Staubli VAL3: s2s7En.pjx

--- s2s7En.pjx ---
Parameters version=s7.9.1 stackSize=5000 millimeterUnit=true
Program file=connectTo.pgx
Program file=getBitAt.pgx
Program file=getByteAt.pgx
Program file=getDBsize.pgx
Program file=getdWordAt.pgx
Program file=getWordAt.pgx
Program file=init.pgx
Program file=ISOConnect.pgx
Program file=isoPDUsize.pgx
Program file=NegotPduLength.pgx
Program file=readArea.pgx
Program file=readDB.pgx
Program file=readme.pgx
Program file=recvISOpacket.pgx
Program file=recvPacket.pgx
Program file=sendPacket.pgx
Program file=setBitAt.pgx
Program file=setByteAt.pgx
Program file=setLastError.pgx
Program file=setWordAt.pgx
Program file=TCPConnect.pgx
Program file=writeArea.pgx
Data file=s2s7En.dtx
Library alias=bitOp path=./Binary7En/Binary7En.pjx
Type name=ISO_PDU_DATA_T path=./ISO_PDU_DATA_T/ISO_PDU_DATA_T.pjx

--- s2s7En.dtx ---
ISO_PDU_DATA_T PDU
  [0]
    num COPT[3]
    S7telegram_T S7telegram
      [0]
        num DATA[240]
        num H[18]
    num TPKT[4]
bool bConnected
public num nAreaCT = 28
public num nAreaDB = 132
public num nAreaMK = 131
public num nAreaPA = 130
public num nAreaPE = 129
public num nAreaTM = 29
num nCC = 208
num nConnType
num nDataBuffer[500]
num nDataSize
num nErrDataRead = 768
num nErrDataWrite = 1024
num nErrISOConnFail = 6
num nErrISOInvPDU = 8
num nErrISONegPDU = 7
num nErrS7Func = 1280
num nErrTCPConnRst = 2
num nErrTCPSend = 4
num nISOPort = 102
num nISO_CR[22]
  [0] = 3
  [3] = 22
  [4] = 17
  [5] = 224
  [9] = 1
  [11] = 192
  [12] = 1
  [13] = 10
  [14] = 193
  [15] = 2
  [16] = 1
  [18] = 194
  [19] = 2
  [20] = 1
  [21] = 2
num nISOheaderSize = 7
public num nLastError
num nLastPDUType
num nLocalTSAP_HI
num nLocalTSAP_LO
num nMaxPduSize = 247
num nMinPduSize = 16
public num nNoErrors
num nPDULength
num nRDsize = 31
num nRecvTimeout = 0.5
num nRemoteTSAP_HI
num nRemoteTSAP_LO
num nS7WLCounter = 28
num nS7WLTimer = 29
num nS7_BI[37]
  [0] = 3
  [3] = 37
  [4] = 2
  [5] = 240
  [6] = 128
  [7] = 50
  [8] = 7
  [11] = 5
  [14] = 8
  [16] = 12
  [18] = 1
  [19] = 18
  [20] = 4
  [21] = 17
  [22] = 67
  [23] = 3
  [25] = 255
  [26] = 9
  [28] = 8
  [29] = 48
  [30] = 65
  [31] = 48
  [32] = 48
  [33] = 48
  [34] = 48
  [35] = 48
  [36] = 65
num nS7_PN[25]
  [0] = 3
  [3] = 25
  [4] = 2
  [5] = 240
  [6] = 128
  [7] = 50
  [8] = 1
  [11] = 4
  [14] = 8
  [17] = 240
  [20] = 1
  [22] = 1
  [24] = 240
num nS7_R[31]
  [0] = 3
  [3] = 31
  [4] = 2
  [5] = 240
  [6] = 128
  [7] = 50
  [8] = 1
  [11] = 5
  [14] = 14
  [17] = 4
  [18] = 1
  [19] = 18
  [20] = 10
  [21] = 16
  [22] = 2
  [27] = 132
num nS7_W[35]
  [0] = 3
  [3] = 31
  [4] = 2
  [5] = 240
  [6] = 128
  [7] = 50
  [8] = 1
  [11] = 5
  [14] = 14
  [17] = 4
  [18] = 1
  [19] = 18
  [20] = 10
  [21] = 16
  [22] = 2
  [27] = 132
  [32] = 4
num nShift = 17
num nTempBuffer
num nWLbit = 1
num nWLbyte = 2
num nWLcounter = 28
num nWLdword = 6
num nWLreal = 8
num nWLtimer = 29
num nWLword = 4
num nWRsize = 35
sio sioTCPclient = {link=Socket\sTcpClient}

--- connectTo.pgx ---
public program connectTo(string x_sIp, num x_nRack, num x_nSlot)
  local num l_nTempDec
  local string l_sRes
  local string l_sTempBin
begin

  //Header begin

  // Create an ISO-on-TCP connection from the controller (client) to the plc (server)
  //
  //Input parameters
  // string x_sIp: ip address of the plc
  // num x_nRack: rack number of the plc (see the hardware configuration in plc's project)
  // num x_nSlot: slot number of the plc (see the hardware configuration in plc's project)

  //Examples
  // call connectTo("127.0.0.1",0,2)
  //
  //History
  // Creation: 24-12-16 - Alessio Villa
  //Header end


  //set connection parameters
  sioCtrl(sioTCPclient,"target",x_sIp)

  nLocalTSAP_HI=1
  nLocalTSAP_LO=0

  //nRemoteTSAP_HI
  l_sTempBin=""
  call bitOp:DecToBin(((nConnType*256)+(x_nRack*32)+x_nSlot),l_sTempBin)
  call bitOp:shiftRight(l_sTempBin,8)
  l_nTempDec=0
  call bitOp:BinToDec(l_sTempBin,l_nTempDec)
  nRemoteTSAP_HI=l_nTempDec

  //nRemoteTSAP_LO
  l_sTempBin=""
  call bitOp:DecToBin(((nConnType*256)+(x_nRack*32)+x_nSlot),l_sTempBin)
  call bitOp:boolAnd(l_sTempBin,"0000000011111111",l_sRes)
  l_nTempDec=0
  call bitOp:BinToDec(l_sRes,l_nTempDec)
  nRemoteTSAP_LO=l_nTempDec

  call setLastError(nNoErrors)
  if !bConnected
    call tcpConnect()
    if nLastError==nNoErrors
      call isoConnect()
      if nLastError==nNoErrors
        //putln("connected to plc!")
        call negotPduLength()
      endIf
    endIf
  endIf

  if nLastError==nNoErrors
    bConnected=true
  endIf

end

--- getBitAt.pgx ---
public program getBitAt(num x_nByteIndex, num x_nBitIndex, num& x_nBuffer[], bool& x_bRes)
  local num l_nResult
  local string l_sByte
  local string l_sMask
  local string l_sResult
begin

  //Header begin

  // This function get the boolean value of the bit number "x_nBitIndex" of the "x_nByteIndex" element (that represent a byte) of the passed array of num (most likely a plc's memory area you read with readArea()).
  //
  //Input parameters
  //
  // num x_nByteIndex: the index of the "x_nBuffer[]" array representing the byte we want to read from (most likely a plc's memory area you read with readArea())
	// num x_nBitIndex: the bit number from 0(LSB) to 7(MSB) in the x_nByteIndex byte, if this value is lower than 0 or higher than 7 x_bRes will be set to false by default.
	// num x_nBuffer[1]: the monodimensional array of num from where we are reading the bit value.
  //
  //Output parameters
  // bool x_bRes: the result, set to "true" if the bit is high, false otherwise.

  //Examples
  //
  // call getBitAt(0,4,l_nRes,l_bRes)
  //
  //History
  // Creation: 24-12-16 - Alessio Villa
  //Header end

  if x_nBitIndex>7
    x_bRes=false
    return
  endIf

  call bitOp:DecToBin(x_nBuffer[x_nByteIndex],l_sByte)
  call bitOp:DecToBin(power(2,x_nBitIndex),l_sMask)
  call bitOp:boolAnd(l_sByte,l_sMask,l_sResult)

  call bitOp:BinToDec(l_sResult,l_nResult)
  if l_nResult>0
    x_bRes=true
  else
    x_bRes=false
  endIf

end

--- getByteAt.pgx ---
public program getByteAt(num x_nByteIndex, num& x_nBuffer[], num& x_nRes)
begin

  //Header begin

  // This function is trivial, it just return in "x_nRes" the "x_nByteIndex" element of the array x_nBuffer (most likely a plc's memory area you read with readArea()).
  //
  //Input parameters
  //
  // num x_nByteIndex: the index of the element in the "x_nBuffer[]" array representing the byte we want to read
	// num x_nBuffer[1]: the monodimensional array of num from where we are reading a byte.

  //Output parameters
  //
  // num x_nRes: where the result is stored

  //Examples
  //
  // 	call getByteAt(12, nDB, l_nRes)
  //
  //History
  // Creation: 24-12-16 - Alessio Villa
  //Header end

  x_nRes=x_nBuffer[x_nByteIndex]

end

--- getDBsize.pgx ---
public program getDBsize(num x_nDBnumber, num& x_nSize)
  local num l_nLength
  local num l_nS7_BI[37]
begin

  //Header begin

  //This function return the size in bytes for a given db
  //
  //Input parameters
  //
  // num x_nDBnumber: the DB number you want to know the size.
  //
  //Output parameters
  //
  // num x_nSize: the variable where the size of the db will be written.
  //
  //Examples
  //
  // call S7:getDBsize(nDBnumber, l_nRes)
  //
  //History
  // Creation: 24-12-16 - Alessio Villa
  //Header end

  call setLastError(nNoErrors)
  x_nSize=0

  //setup the telegram
  getData("nS7_BI",l_nS7_BI)

  l_nS7_BI[31]=round((x_nDBnumber/10000)+48)
  x_nDBnumber=round(x_nDBnumber%10000)

  l_nS7_BI[32]=round((x_nDBnumber/1000)+48)
  x_nDBnumber=round(x_nDBnumber%1000)

  l_nS7_BI[33]=round((x_nDBnumber/100)+48)
  x_nDBnumber=round(x_nDBnumber%100)

  l_nS7_BI[34]=round((x_nDBnumber/10)+48)
  x_nDBnumber=round(x_nDBnumber%10)

  l_nS7_BI[35]=round((x_nDBnumber)+48)

  call sendPacket(l_nS7_BI,size(l_nS7_BI))
  if nLastError==nNoErrors
    call recvISOpacket(l_nLength)
    //26 is the minimum expected
    if l_nLength>=26
      //if ((PDU.H[37]==0x00) && (PDU.H[38]==0x00) && (PDU.H[39]==0xFF))
      if PDU.S7telegram.DATA[2]==0 or PDU.S7telegram.DATA[3]==0 or PDU.S7telegram.DATA[4]==255
        x_nSize=PDU.S7telegram.DATA[48]
        x_nSize=x_nSize*power(2,8)+PDU.S7telegram.DATA[49]
      else
        call setLastError(nErrS7Func)
      endIf
    else
      call setLastError(nErrISOInvPDU)
    endIf
  else
    call setLastError(nErrTCPSend)
  endIf

end

--- getdWordAt.pgx ---
public program getDwordAt(num x_nByteIndex, num& x_nBuffer[], num& x_nRes)
begin

  //Header begin

  //This function return in "x_nRes" the value of the double word composed by four bytes starting from "x_nByteIndex" element of the array x_nBuffer (most likely a plc's memory area you read with readArea()).
  //The first byte is the lower part of the word (Big Endian)
  //
  //Input parameters
  //
  //num x_nByteIndex: the index of the element in the "x_nBuffer[]" array representing the starting byte of the double word we want to read
	//num x_nBuffer[1]: the monodimensional array of num from where we are reading a double word.
  //
  //Output parameters
  //
  // num x_nRes: where the result is stored.
  //
  //Examples
  //
  // 	call getDWordAt(7, nDB, l_nRes)
  //
  //History
  // Creation: 24-12-16 - Alessio Villa
  //Header end

  x_nRes=x_nBuffer[x_nByteIndex]*power(2,24)+x_nBuffer[x_nByteIndex+1]*power(2,16)+x_nBuffer[x_nByteIndex+2]*power(2,8)+x_nBuffer[x_nByteIndex+3]

end

--- getWordAt.pgx ---
public program getWordAt(num x_nByteIndex, num& x_nBuffer[], num& x_nRes)
begin

  //Header begin

  //This function return in "x_nRes" the value of the word composed by two bytes starting from "x_nByteIndex" element of the array x_nBuffer (most likely a plc's memory area you read with readArea()).
  //The first byte is the lower part of the word (Big Endian)
  //
  //Input parameters
  //
  //num x_nByteIndex: the index of the element in the "x_nBuffer[]" array representing the starting byte of the double word we want to read
	//num x_nBuffer[1]: the monodimensional array of num from where we are reading a double word.
  //
  //Output parameters
  //
  // num x_nRes: where the result is stored.
  //
  //Examples
  //
  // 	call getWordAt(3, nDB, l_nRes)
  //
  //History
  // Creation: 24-12-16 - Alessio Villa
  //Header end

  x_nRes=x_nBuffer[x_nByteIndex]*power(2,8)+x_nBuffer[x_nByteIndex+1]

end

--- init.pgx ---
public program init(sio& x_sTCPclient)
begin

  //Header begin
  // This function initialize the library.
  //Use it once at the beginning of your VAL3 application.
  //
  //Input parameters
  //
  //x_sTCPclient: the sio variable linked with the TCP client socket you must define on your controller.
  //
  //Output parameters
  //
  //Examples
  //
  //  call S7:init(sTcpClient)
  //History
  // Creation: 24-12-16 - Alessio Villa
  //Header end

  sioLink(sioTCPclient,x_sTCPclient)
  sioCtrl(sioTCPclient,"port",nISOPort)
  sioCtrl(sioTCPclient,"timeout",nRecvTimeout)
  sioCtrl(sioTCPclient,"endOfString",13)
  sioCtrl(sioTCPclient,"clients",1)
  sioCtrl(sioTCPclient,"nagle",false)


  nLocalTSAP_HI=1
  nLocalTSAP_LO=0
  nRemoteTSAP_HI=1
  nRemoteTSAP_LO=2

  bConnected=false
  //PG connection type
  nConnType=1
  call setLastError(nNoErrors)
  nPDULength=0
  nRecvTimeout=0.5

end

--- ISOConnect.pgx ---
program isoConnect()
  local num l_nLength
begin

  nISO_CR[16]=nLocalTSAP_HI
  nISO_CR[17]=nLocalTSAP_LO
  nISO_CR[20]=nRemoteTSAP_HI
  nISO_CR[21]=nRemoteTSAP_LO

  //if sioSet(sTCPclient, nISO_CR) == size(nISO_CR)
  call sendPacket(nISO_CR,size(nISO_CR))
  if nLastError==nNoErrors
    call recvISOpacket(l_nLength)
    //15 = 22 (sizeof CC telegram) - 7 (sizeof Header)
    if nLastError==nNoErrors and l_nLength==15
      //it was a connection confirm?
      if nLastPDUType!=nCC
        call setLastError(nErrISOInvPDU)
      endIf
    endIf
  else
    call setLastError(nErrISOConnFail)
  endIf

end

--- isoPDUsize.pgx ---
program isoPDUsize(num& x_nSize)
begin

  x_nSize=PDU.TPKT[2]
  x_nSize=x_nSize*256+PDU.TPKT[3]

end

--- NegotPduLength.pgx ---
program negotPduLength()
  local num l_nLength
begin

  //if sioSet(sTCPclient, nS7_PN) == size(nS7_PN)
  call sendPacket(nS7_PN,size(nS7_PN))
  if nLastError==nNoErrors
    call recvISOpacket(l_nLength)
    if nLastError==nNoErrors
      //20 = size of Negotiate Answer, then check S7 Error
      //if l_nLength==20 and PDU.H[27]==0 and PDU.H[28]==0
      if l_nLength==20 and PDU.S7telegram.H[10]==0 and PDU.S7telegram.H[11]==0
        nPDULength=PDU.S7telegram.DATA[0]
        nPDULength=nPDULength*power(2,8)+PDU.S7telegram.DATA[1]
        if nPDULength>0
          //put("PDU length negotiated:")
          //put(nPDULength)
          //putln(" bytes")
        else
          call setLastError(nErrISONegPDU)
        endIf
      else
        call setLastError(nErrISONegPDU)
      endIf
    else
      call setLastError(nErrISONegPDU)
    endIf
  else
    call setLastError(nErrISONegPDU)
  endIf


end

--- readArea.pgx ---
public program readArea(num x_nIdArea, num x_nDBnumber, num x_nStartAt, num x_nQty, num& x_nBuffer[])
  local num l_Address
  local num l_nElementsNum
  local num l_nIndex
  local num l_nLength
  local num l_nMaxElements
  local num l_nOffs
  local num l_nS7R[31]
  local num l_nSizeReq
  local num l_nTempDec
  local num l_nToIndex
  local num l_nTotElements
  local num l_nWordSize
  local string l_sRes
  local string l_sTempBin
begin

  //Header begin

  //This function read a memory area from the PLC starting from "x_nStartAt" byte and for a "x_nQty" number of bytes.
  //The result is stored in a "num" array where each element is a byte of the memory area read.
  //
  //Input parameters
  //
  //num x_nIdArea: the PLC's memory area identifier (you'll find several identifier as public members of the library with the suffix "nArea").
	//num x_nDBnumber: the DB number you're reading from (this parameter is not important if you're not reading a db...but in VAL3 there's no possibility to overload functions so we must pass it the same to this function!).
	//num x_nStartAt:: the byte adddress you want start to read from.
	//num x_nQty: the amount of bytes you want to read.
  //
  //Output parameters
  // num x_nBuffer[1]:  a monodimensional array where the area read is stored. If the size of this buffer is smaller than "x_nQty" only "size(x_nBuffer[])" will be read .
  //
  //Examples
  //
  // call S7:readArea(S7:nAreaDB,nDBread,2,1,l_nRes)
  //
  //History
  // Creation: 24-12-16 - Alessio Villa
  //Header end

  l_nOffs=0
  l_nWordSize=1

  call setLastError(nNoErrors)

  if size(x_nBuffer)<x_nQty
    //small buffer
    x_nQty=size(x_nBuffer)
  endIf

  if x_nIdArea==nAreaCT or x_nIdArea==nAreaTM
    l_nWordSize=2
  endIf

  //18 is the reply header size
  l_nMaxElements=(nPDULength-18)/l_nWordSize
  l_nTotElements=x_nQty

  while l_nTotElements>0 and nLastError==nNoErrors

    l_nElementsNum=l_nTotElements
    if l_nElementsNum>l_nMaxElements
      l_nElementsNum=l_nMaxElements
    endIf
    //calc request size
    l_nSizeReq=l_nElementsNum*l_nWordSize

    //setup the telegram!
    getData("nS7_R",l_nS7R)

    //set area number
    l_nS7R[27]=x_nIdArea
    if x_nIdArea==nAreaDB
      //set db number
      l_sTempBin=""
      call bitOp:DecToBin(x_nDBnumber,l_sTempBin)
      call bitOp:shiftRight(l_sTempBin,8)
      l_nTempDec=0
      call bitOp:BinToDec(l_sTempBin,l_nTempDec)
      l_nS7R[25]=l_nTempDec
      l_sTempBin=""
      call bitOp:DecToBin(x_nDBnumber,l_sTempBin)
      l_sRes=""
      call bitOp:boolAnd(l_sTempBin,"0000000011111111",l_sRes)
      l_nTempDec=0
      call bitOp:BinToDec(l_sRes,l_nTempDec)
      l_nS7R[26]=l_nTempDec
    endIf

    // Adjusts Start and word length
    if x_nIdArea==nAreaCT or x_nIdArea==nAreaTM
      l_Address=x_nStartAt
      if x_nIdArea==nAreaCT
        l_nS7R[22]=nWLcounter
      else
        l_nS7R[22]=nWLtimer
      endIf
    else
      //shift left 3 bit
      l_Address=x_nStartAt*power(2,3)
    endIf

    //number of elements
    l_nS7R[23]=l_nElementsNum*power(2,8)
    l_nS7R[24]=l_nElementsNum
    //address in plc
    l_sTempBin=""
    call bitOp:DecToBin(l_Address,l_sTempBin)
    l_sRes=""
    call bitOp:boolAnd(l_sTempBin,"0000000011111111",l_sRes)
    l_nTempDec=0
    call bitOp:BinToDec(l_sRes,l_nTempDec)
    l_nS7R[30]=l_nTempDec
    call bitOp:shiftRight(l_sTempBin,8)

    l_sRes=""
    call bitOp:boolAnd(l_sTempBin,"0000000011111111",l_sRes)
    l_nTempDec=0
    call bitOp:BinToDec(l_sRes,l_nTempDec)
    l_nS7R[29]=l_nTempDec
    call bitOp:shiftRight(l_sTempBin,8)

    l_sRes=""
    call bitOp:boolAnd(l_sTempBin,"0000000011111111",l_sRes)
    l_nTempDec=0
    call bitOp:BinToDec(l_sRes,l_nTempDec)
    l_nS7R[28]=l_nTempDec

    //send the telegram!
    call sendPacket(l_nS7R,nRDsize)
    if nLastError==nNoErrors
      call recvISOpacket(l_nLength)
      if nLastError==nNoErrors
        if l_nLength>=18
          //if ((Length-18==SizeRequested) && (PDU.H[31]==0xFF))
          if l_nLength-18==l_nSizeReq and PDU.S7telegram.H[14]==255
            //copy data in the target buffer
            l_nIndex=0
            if size(x_nBuffer)-l_nOffs<size(PDU.S7telegram.DATA)
              l_nToIndex=size(x_nBuffer)-l_nOffs-1
            else
              l_nToIndex=size(PDU.S7telegram.DATA)-1
            endIf
            for l_nIndex=0 to l_nToIndex
              x_nBuffer[l_nOffs+l_nIndex]=PDU.S7telegram.DATA[l_nIndex]
            endFor
            l_nOffs=l_nOffs+l_nSizeReq
          else
            call setLastError(nErrDataRead)
          endIf
        else
          call setLastError(nErrISOInvPDU)
        endIf
      else
        //error detected
      endIf
    else
      call setLastError(nErrTCPSend)
    endIf

    l_nTotElements=l_nTotElements-l_nElementsNum
    x_nStartAt=x_nStartAt+l_nElementsNum*l_nWordSize

  endWhile

end

--- readDB.pgx ---
public program readDB(num x_nDBnumber, num& x_nDB[])
  local num l_nLength
begin

  //Header begin

  // This function is a convenient wrapper of "readArea" useful to read a whole DB from the PLC.
  //
  //Input parameters
  //
  // num x_nDBnumber:the DB number you want to read
  //
  //Output parameters
  //
  // num x_nDB[1]:a monodimensional array of "num" where the db is stored. The size of this buffer will be resized to match exactly the db's size , for this reason x_nDB[] MUST BE A GLOBAL VARIABLE.
  //
  //Examples
  //
  // call S7:readDB(nDBnumber, nDB)
  //
  //History
  // Creation: 24-12-16 - Alessio Villa
  //Header end

  call getDBsize(x_nDBnumber,l_nLength)

  if nLastError==nNoErrors
    resize(x_nDB,1,l_nLength)
    call readArea(nAreaDB,x_nDBnumber,0,l_nLength,x_nDB)
  endIf

end

--- readme.pgx ---
program readme()
begin

  //Title: S2S Library (Staubli to Siemens)
  //General description:  S2S is a minimal VAL3 porting of the "S7_micro_client" class of the SNAP7 library (Copyright (C) 2013, Davide Nardella, http://snap7.sourceforge.net/).
  //It allows the read/write communication from a Staubli controller to a Siemens PLC over a standard ethernet TCP/IP connection.
  //
  //Hardware required: Siemens PLC's S7 300/400/WinAC or S7 1200/1500 (see the complete documentation here: https://github.com/alejho/S2S)
  //
  //VAL3 options: 7.9.1
  //
  //Library version: 7.9.1.1
  //
  //Public variables: nAreaCT, nAreaDB, nAreaMK, nAreaPA, nAreaPE, nAreaTM, nLastError, nNoErrors
  //
  //

  //Miscellaneous: Since the snap7 are released under lgplv3 license and this is a derivative work, this library is also released un lgplv3 license.
  //You should have received a copy of the GNU General Public License and a copy of Lesser GNU General Public License along with S2S, if not, see  http://www.gnu.org/licenses/
  //For licensing reasons the library must be publicly available here: https://github.com/alejho/S2S where you can find the most up-to-date version and a full documentation of this library.
  //
  //Contact the author (a.villa@staubli.com) for support and information.
  //
  //Keywords: Siemens PLC Ethernet
end

--- recvISOpacket.pgx ---
program recvISOpacket(num& x_nLength)
  local num i
  local bool l_bDone
begin

  nLastError=0

  while (nLastError==nNoErrors and !l_bDone)
    // Get TPKT (4 bytes)
    call recvPacket(PDU.TPKT,4)
    if nLastError==nNoErrors
      call isoPDUsize(x_nLength)
      if x_nLength==7
        //only TPKT+COTP(7bytes)...skip next 3 bytes and receive another packet
        call recvPacket(PDU.COPT,3)
      elseIf x_nLength>nMaxPduSize or x_nLength<nMinPduSize
        //wrong size!
        call setLastError(nErrISOInvPDU)
      else
        //valid length !=7 && >16 && <247...done!
        l_bDone=true
      endIf
    endIf
  endWhile

  if nLastError==nNoErrors
    // Skip remaining 3 COTP bytes
    call recvPacket(PDU.COPT,3)
    nLastPDUType=PDU.COPT[1]
    x_nLength=x_nLength-nISOheaderSize
    call recvPacket(nDataBuffer,x_nLength)
    for i=0 to size(PDU.S7telegram.H)-1
      PDU.S7telegram.H[i]=nDataBuffer[i]
    endFor
    for i=0 to size(PDU.S7telegram.DATA)-1
      PDU.S7telegram.DATA[i]=nDataBuffer[i+size(PDU.S7telegram.H)]
    endFor
  else
    clearBuffer(sioTCPclient)
  endIf

end

--- recvPacket.pgx ---
program recvPacket(num& x_nBuff[], num x_nSize)
begin

  resize(nTempBuffer,1,1)
  nTempBuffer=0
  resize(nTempBuffer,1,x_nSize)

  if sioGet(sioTCPclient,nTempBuffer)!=x_nSize
    call setLastError(nErrTCPConnRst)
  endIf

  getData("nTempBuffer",x_nBuff)

end

--- sendPacket.pgx ---
program sendPacket(num& x_nBuff[], num x_nSize)
  local num l_nIndex
begin

  resize(nTempBuffer,1,1)
  nTempBuffer=0
  if x_nSize>0
    resize(nTempBuffer,1,x_nSize)
  else
    call setLastError(nErrTCPSend)
    return
  endIf

  for l_nIndex=0 to x_nSize-1
    nTempBuffer[l_nIndex]=x_nBuff[l_nIndex]
  endFor

  //if the server is down this function is blocking this:
  //if watch(sioSet(sTCPclient, nTempBuffer) == size(nTempBuffer), nRecvTimeout)
  //...doesnt work because sioSet is blocked!...maybe we need to do this in a separate task and wait a response from this task!

  if sioSet(sioTCPclient,nTempBuffer)!=size(nTempBuffer)
    call setLastError(nErrTCPConnRst)
  endIf

end

--- setBitAt.pgx ---
public program setBitAt(num x_nByteIndex, num x_nBitIndex, bool x_bBit, num& x_nBuffer[])
begin

  //Header begin

  // This function set to "x_bBit" the boolean value of the bit number "x_nBitIndex" of the "x_nByteIndex" element (that represent a byte) of the passed array of num.
  //
  //Input parameters
  //
  //num x_nByteIndex: the index of the "x_nBuffer[]" array representing the byte we want to set.
	//num x_nBitIndex: the bit number from 0(LSB) to 7(MSB) in the x_nByteIndex byte, if this value is lower than 0 or higher than 7 this function will have no effetcs.
	//num x_bBit: the boolean value we want to set.
  //
  //Output parameters
  //
  // num x_nBuffer[1]: the monodimensional array of num from we are writing the bit value (most likely a plc's memory area we are about to write with writeArea).
  //
  //Examples
  //
  // call setBitAt(0, 3, true, nPlcWriteBuffer)
  //
  //History
  // Creation: 24-12-16 - Alessio Villa
  //Header end

  if x_nBitIndex>7
    return
  endIf

  if x_bBit
    x_nBuffer[x_nByteIndex]=bOr(power(2,x_nBitIndex),x_nBuffer[x_nByteIndex])
  else
    x_nBuffer[x_nByteIndex]=bAnd(power(2,8)-power(2,x_nBitIndex)-1,x_nBuffer[x_nByteIndex])
  endIf

end

--- setByteAt.pgx ---
public program setByteAt(num x_nByteIndex, num x_nByte, num& x_nBuffer[])
  local num l_nHIword
  local num l_nLOword
  local string l_sBinWord
  local string l_sTempBinByte
begin

  //Header begin

  //This function is trivial, it just set to "x_nByte" the "x_nByteIndex" element of the array x_nBuffer.
  //
  //Input parameters
  //
  //num x_nByteIndex: the index of the element in the "x_nBuffer[]" array representing the byte we want to read.
	//num x_nRes: the byte value we want to set.
  //
  //Output parameters
  //
  //num x_nBuffer[1]: the monodimensional array of num where we are writing a byte (most likely a plc's memory area we are about to write with writeArea).
  //
  //Examples
  //
  //call S7:setWordAt(0,231,l_nLocalByte)
  //
  //History
  // Creation: 24-12-16 - Alessio Villa
  //Header end

  if x_nByte<0 or x_nByte>255
    x_nBuffer[x_nByteIndex]=0
  endIf

  x_nBuffer[x_nByteIndex]=x_nByte

end

--- setLastError.pgx ---
program setLastError(num x_nError)
begin

  //Header begin

  // Describe functionality and purpose
  //
  //Input parameters
  // type param1: description (role, possible values,...)
  // param1 description (continued)
  // param1 description (continued)
  // type param2: description (role, possible values,...)
  // type param3: description (role, possible values,...)
  // ...
  //
  //Output parameters
  // type param1: description (role, possible values,...)
  // type param2: description (role, possible values,...)
  // type param3: description (role, possible values,...)
  // ...
  //
  //Examples
  // call examples (for public programs mostly)
  //
  //History
  // Creation: DD-MM-YY - AUTHOR NAME
  // Modification: DD-MM-YY - AUTHOR NAME - Description of modification
  // description of modification (continued)
  // description of modification (continued)
  // Modification: DD-MM-YY - AUTHOR NAME - Description of modification
  //Header end

  nLastError=x_nError

end

--- setWordAt.pgx ---
public program setWordAt(num x_nByteIndex, num x_nWord, num& x_nBuffer[])
  local num l_nHIword
  local num l_nLOword
  local string l_sBinWord
  local string l_sTempBinByte
begin

  //Header begin

  // This function set to "x_nWord" the value of the word composed by two bytes starting from "x_nByteIndex" element of the array x_nBuffer (most likely a plc's memory area we are about to write with writeArea).
  // This will be done according to the Big Endian notation used in Siemens.
  //
  //Input parameters
  //
  //num x_nByteIndex: the index of the element in the "x_nBuffer[]" array representing the starting byte of the word we want to read.
	//num x_nRes: the word value we want to set.
  //
  //Output parameters
  //
  //num x_nBuffer[1]: the monodimensional array of num where we are writing a word (most likely a plc's memory area we are about to write with writeArea).
  //
  //Examples
  //
  // call setWordAt(0,554,l_nLocalWord)
  //
  //History
  // Creation: 24-12-16 - Alessio Villa
  //Header end

  //gestione del segno???
  if x_nWord<0 or x_nWord>power(2,16)-1
    x_nBuffer[x_nByteIndex]=0
    x_nBuffer[x_nByteIndex+1]=0
    return
  endIf

  l_sBinWord=""
  call bitOp:BitWord(x_nWord,l_sBinWord)
  call bitOp:shiftRight(l_sBinWord,8)
  call bitOp:BinToDec(l_sBinWord,l_nLOword)

  l_sBinWord=""
  call bitOp:BitWord(x_nWord,l_sBinWord)
  call bitOp:boolAnd(l_sBinWord,"0000000011111111",l_sTempBinByte)
  call bitOp:BinToDec(l_sTempBinByte,l_nHIword)

  x_nBuffer[x_nByteIndex]=l_nLOword
  x_nBuffer[x_nByteIndex+1]=l_nHIword

end

--- TCPConnect.pgx ---
program tcpConnect()
begin

  //there's nothing like client.connect in val3 socket...it's the os to handle this stuff when you try to write something!

end

--- writeArea.pgx ---
public program writeArea(num x_nIdArea, num x_nDBnumber, num& x_nBuffer[], num x_nStartAt, num x_nQty)
  local num l_Address
  local bool l_bLoop
  local num l_nDataSize
  local num l_nElementsNum
  local num l_nIndex
  local num l_nIsoSize
  local num l_nLength
  local num l_nMaxElements
  local num l_nOffs
  local num l_nS7W[35]
  local num l_nTempDec
  local num l_nTotElements
  local num l_nWordSize
  local string l_sRes
  local string l_sTempBin
begin

  //Header begin

  // This function write in a given PLC memory's area the content of the passed array of num, starting from a gven byte and for a given amount of bytes.
  //
  //Input parameters
  //
  //num x_nIdArea: the PLC's memory area identifier (you'll find several identifier as public members of the library with the suffix "nArea").
	//num x_nDBnumber: the DB number you're writing to (this parameter is not important if you're not writing a db...but in VAL3 there's no possibility to overload functions so we must pass it the same to this function!).
	//num x_nBuffer[1]:  a monodimensional array where representing the memory area we want to write. If the size of this buffer is smaller than "x_nQty" only "size(x_nBuffer[])" will be written .
	//num x_nStartAt: the byte address you want start to write from.
	//num x_nQty: the amount of bytes you want to write.
  //
  //Examples
  //
  //call S7:writeArea(S7:nAreaDB, nDBnumber, nSampleBuffer, 0, size(nSampleBuffer))
  //
  //History
  //
  // Creation: 24-12-16 - Alessio Villa
  //Header end

  l_nOffs=0
  l_nWordSize=1

  call setLastError(nNoErrors)

  if x_nIdArea==nAreaCT or x_nIdArea==nAreaTM
    l_nWordSize=2
  endIf

  l_nMaxElements=(nPDULength-size(nS7_W))/l_nWordSize
  l_nTotElements=x_nQty

  while l_nTotElements>0 and nLastError==nNoErrors

    l_nElementsNum=l_nTotElements
    if l_nElementsNum>l_nMaxElements
      l_nElementsNum=l_nMaxElements
    endIf

    l_nDataSize=l_nElementsNum*l_nWordSize
    l_nIsoSize=size(nS7_W)+l_nDataSize

    //setup the telegram
    getData("nS7_W",l_nS7W)

    //telegram size high byte
    l_sTempBin=""
    call bitOp:DecToBin(l_nIsoSize,l_sTempBin)
    call bitOp:shiftRight(l_sTempBin,8)
    l_nTempDec=0
    call bitOp:BinToDec(l_sTempBin,l_nTempDec)
    l_nS7W[2]=l_nTempDec

    //telegram size low byte
    l_sTempBin=""
    call bitOp:DecToBin(l_nIsoSize,l_sTempBin)
    l_sRes=""
    call bitOp:boolAnd(l_sTempBin,"0000000011111111",l_sRes)
    l_nTempDec=0
    call bitOp:BinToDec(l_sTempBin,l_nTempDec)
    l_nS7W[3]=l_nTempDec

    //data length high byte
    l_nLength=l_nDataSize+4
    l_sTempBin=""
    call bitOp:DecToBin(l_nLength,l_sTempBin)
    call bitOp:shiftRight(l_sTempBin,8)
    l_nTempDec=0
    call bitOp:BinToDec(l_sTempBin,l_nTempDec)
    l_nS7W[15]=l_nTempDec

    //data length low bytes
    l_sTempBin=""
    call bitOp:DecToBin(l_nLength,l_sTempBin)
    l_sRes=""
    call bitOp:boolAnd(l_sTempBin,"0000000011111111",l_sRes)
    l_nTempDec=0
    call bitOp:BinToDec(l_sTempBin,l_nTempDec)
    l_nS7W[16]=l_nTempDec

    //function id
    l_nS7W[17]=5
    //plc memory area
    l_nS7W[27]=x_nIdArea
    if x_nIdArea==nAreaDB
      //db number high byte
      l_sTempBin=""
      call bitOp:DecToBin(x_nDBnumber,l_sTempBin)
      call bitOp:shiftRight(l_sTempBin,8)
      l_nTempDec=0
      call bitOp:BinToDec(l_sTempBin,l_nTempDec)
      l_nS7W[25]=l_nTempDec
      //db number low byte
      l_sTempBin=""
      call bitOp:DecToBin(x_nDBnumber,l_sTempBin)
      l_sRes=""
      call bitOp:boolAnd(l_sTempBin,"0000000011111111",l_sRes)
      l_nTempDec=0
      call bitOp:BinToDec(l_sTempBin,l_nTempDec)
      l_nS7W[26]=l_nTempDec
    endIf
    // Adjusts Start and word length
    if x_nIdArea==nAreaCT or x_nIdArea==nAreaTM
      l_Address=x_nStartAt
      l_nLength=l_nDataSize
      if x_nIdArea==nAreaCT
        l_nS7W[22]=nS7WLCounter
      else
        l_nS7W[22]=nS7WLTimer
      endIf
    else
      //shift left 3 bit
      l_Address=x_nStartAt*power(2,3)
      //shift left 3 bit
      l_nLength=l_nDataSize*power(2,3)
    endIf

    l_nS7W[23]=l_nElementsNum*power(2,8)
    l_nS7W[24]=l_nElementsNum
    //address in plc
    l_sTempBin=""
    call bitOp:DecToBin(l_Address,l_sTempBin)
    l_sRes=""
    call bitOp:boolAnd(l_sTempBin,"0000000011111111",l_sRes)
    l_nTempDec=0
    call bitOp:BinToDec(l_sRes,l_nTempDec)
    l_nS7W[30]=l_nTempDec
    call bitOp:shiftRight(l_sTempBin,8)

    l_sRes=""
    call bitOp:boolAnd(l_sTempBin,"0000000011111111",l_sRes)
    l_nTempDec=0
    call bitOp:BinToDec(l_sRes,l_nTempDec)
    l_nS7W[29]=l_nTempDec
    call bitOp:shiftRight(l_sTempBin,8)

    l_sRes=""
    call bitOp:boolAnd(l_sTempBin,"0000000011111111",l_sRes)
    l_nTempDec=0
    call bitOp:BinToDec(l_sRes,l_nTempDec)
    l_nS7W[28]=l_nTempDec

    //length high byte
    l_sTempBin=""
    call bitOp:DecToBin(l_nLength,l_sTempBin)
    call bitOp:shiftRight(l_sTempBin,8)
    l_nTempDec=0
    call bitOp:BinToDec(l_sTempBin,l_nTempDec)
    l_nS7W[33]=l_nTempDec
    //legth low byte
    l_sTempBin=""
    call bitOp:DecToBin(l_nLength,l_sTempBin)
    l_sRes=""
    call bitOp:boolAnd(l_sTempBin,"0000000011111111",l_sRes)
    l_nTempDec=0
    call bitOp:BinToDec(l_sTempBin,l_nTempDec)
    l_nS7W[34]=l_nTempDec
    //copy data to be sent in the telegram from where i finished in the previous iteration
    l_bLoop=true
    l_nIndex=0
    while l_bLoop
      PDU.S7telegram.DATA[l_nIndex]=x_nBuffer[l_nOffs+l_nIndex]
      l_nIndex=l_nIndex+1
      if l_nIndex>=size(PDU.S7telegram.DATA) or (l_nIndex+l_nOffs)>=size(x_nBuffer)
        l_bLoop=false
      endIf
    endWhile
    //send header
    call sendPacket(l_nS7W,size(nS7_W))
    //send data
    call sendPacket(PDU.S7telegram.DATA,l_nIsoSize-size(nS7_W))
    if nLastError==nNoErrors
      call recvISOpacket(l_nLength)
      if nLastError==nNoErrors
        //15 is expected here!
        if l_nLength==15
          if PDU.S7telegram.H[10]!=0 or PDU.S7telegram.H[11]!=0 or PDU.S7telegram.H[14]!=255
            call setLastError(nErrDataWrite)
          endIf
        else
          call setLastError(nErrISOInvPDU)
        endIf
      endIf
    else
      //error while sending packet
      call setLastError(nErrTCPSend)
    endIf

    l_nOffs=l_nOffs+l_nDataSize
    l_nTotElements=l_nTotElements-l_nElementsNum
    x_nStartAt=x_nStartAt+l_nElementsNum*l_nWordSize

  endWhile
end
